// Mitsubishi GX Works2 project: PLC PROJECT   PLC: Q03UDE

PROGRAM MAIN
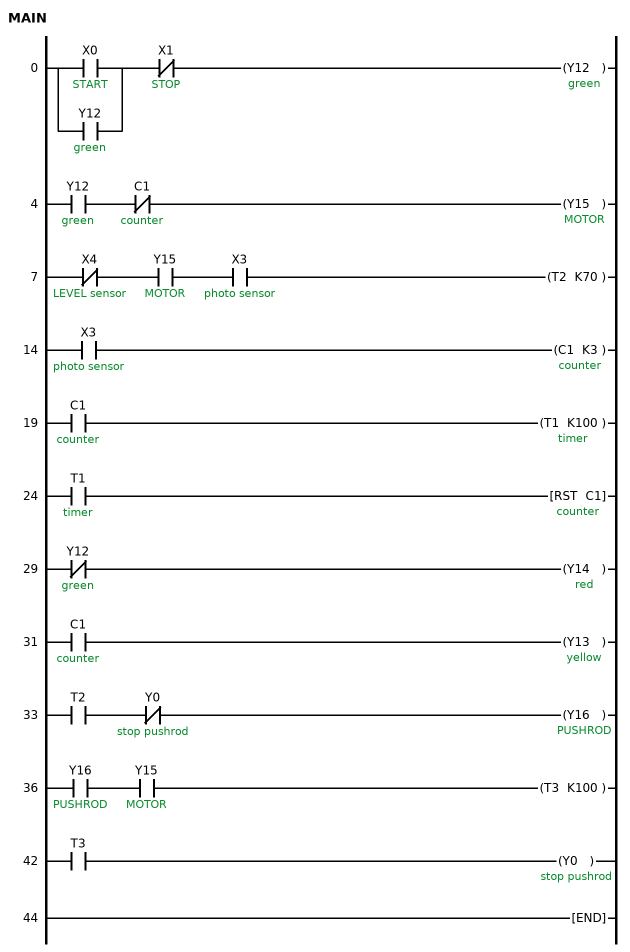
0     LD      X0  ; START
      OR      Y12  ; green
      ANI     X1  ; STOP
      OUT     Y12  ; green
4     LD      Y12  ; green
      ANI     C1  ; counter
      OUT     Y15  ; MOTOR
7     LDI     X4  ; LEVEL sensor
      AND     Y15  ; MOTOR
      AND     X3  ; photo sensor
      OUT     T2 K70
14    LD      X3  ; photo sensor
      OUT     C1 K3  ; counter
19    LD      C1  ; counter
      OUT     T1 K100  ; timer
24    LD      T1  ; timer
      RST     C1  ; counter
29    LDI     Y12  ; green
      OUT     Y14  ; red
31    LD      C1  ; counter
      OUT     Y13  ; yellow
33    LD      T2
      ANI     Y0  ; stop pushrod
      OUT     Y16  ; PUSHROD
36    LD      Y16  ; PUSHROD
      AND     Y15  ; MOTOR
      OUT     T3 K100
42    LD      T3
      OUT     Y0  ; stop pushrod
44    END
END_PROGRAM

// device comments not shown above
X2  ; stop
Y10  ; motor
Y11  ; push rod
T4  ; Timer
